PROGRAM PRG_RCC
VAR
	RCC_VRC_01_OPEN_OK : BOOL;
	RCC_VRC_02_OPEN_OK : BOOL;
	RCC_VRC_03_OPEN_OK : BOOL;
	RCC_VRC_04_OPEN_OK : BOOL;
	
END_VAR

RCC_GCP_01(PG=>);

RCC_STC_01(
	iScale:= , 
	fTemp=> , 
	);
(* Valve can open only when CRIX-RCC-VRC-02 and 03 are closed*)		
RCC_VRC_01_OPEN_OK := ( RCC_VRC_02.iq_stValve.i_xClsLS AND NOT RCC_VRC_02.iq_stValve.q_xOPN_DO ) AND
                                    ( RCC_VRC_03.iq_stValve.i_xClsLS AND NOT RCC_VRC_03.iq_stValve.q_xOPN_DO ) ;
						   
RCC_VRC_01(i_xExtILK_OK := RCC_VRC_01_OPEN_OK, 
                i_xOverrideMode := xSystemOverrideMode_RCC, 
                 iq_stValve=> );

(* Valve can open only when CRIX-RCC-VRC-01 and 04 are closed*)				 
RCC_VRC_02_OPEN_OK := ( RCC_VRC_01.iq_stValve.i_xClsLS AND NOT RCC_VRC_01.iq_stValve.q_xOPN_DO ) AND
                                    ( RCC_VRC_04.iq_stValve.i_xClsLS AND NOT RCC_VRC_04.iq_stValve.q_xOPN_DO );
						   
RCC_VRC_02(i_xExtILK_OK := RCC_VRC_02_OPEN_OK, 
                i_xOverrideMode := xSystemOverrideMode_RCC, 
                 iq_stValve=> );				 

(* Valve can open only when CRIX-RCC-GCP-01 reading <10 Torr and CRIX-RCC-VRC-01 and 04 are closed*)							 
RCC_VRC_03_OPEN_OK := (RCC_GCP_01.PG.rPRESS < 10 and RCC_GCP_01.PG.xPRESS_OK ) AND
                                 ( RCC_VRC_01.iq_stValve.i_xClsLS AND NOT RCC_VRC_01.iq_stValve.q_xOPN_DO ) AND
                                              ( RCC_VRC_04.iq_stValve.i_xClsLS AND NOT RCC_VRC_04.iq_stValve.q_xOPN_DO );				 

RCC_VRC_03(i_xExtILK_OK := RCC_VRC_03_OPEN_OK, 
                i_xOverrideMode := xSystemOverrideMode_RCC, 
                 iq_stValve=> );

(* Valve can open only when CRIX-RCC-VRC-02 and 03 are closed*)		
RCC_VRC_04_OPEN_OK := ( RCC_VRC_02.iq_stValve.i_xClsLS AND NOT RCC_VRC_02.iq_stValve.q_xOPN_DO ) AND
                                      ( RCC_VRC_03.iq_stValve.i_xClsLS AND NOT RCC_VRC_03.iq_stValve.q_xOPN_DO ) ;

RCC_VRC_04(i_xExtILK_OK := RCC_VRC_04_OPEN_OK, 
                i_xOverrideMode := xSystemOverrideMode_RCC, 
                 iq_stValve=> );

END_PROGRAM

(* stored: Version 1.1.0.1, ProductVersion 3.1.4022.18
   POU PRG_RCC: Id {89e03fdd-ce79-4cd4-8b3e-f2ec4b282ec5}, SpecialFunc None *)
